FUNCTION_BLOCK FB_2001_cocktail
VAR_INPUT
	execute: BOOL;
END_VAR
VAR
	TIMERDONE: BOOL;
END_VAR

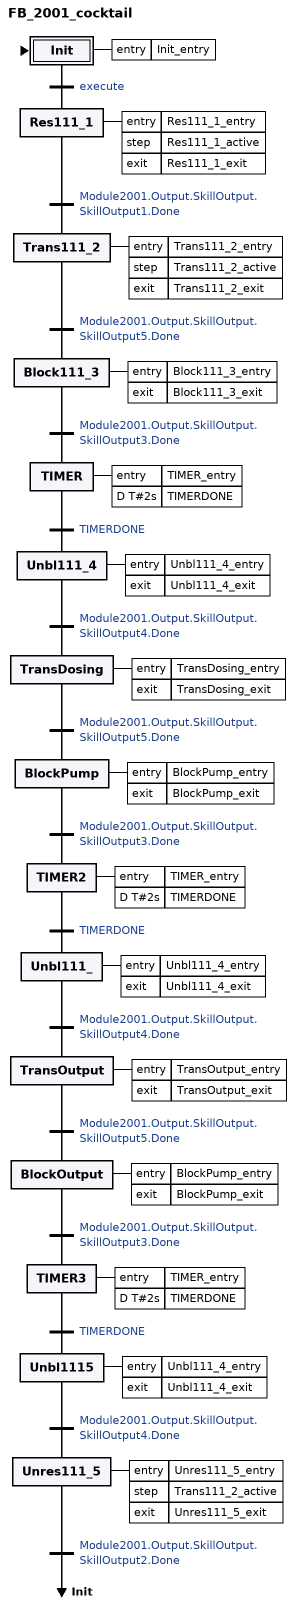
INITIAL_STEP Init:
    Init_entry(P1);  // entry action
END_STEP
TRANSITION FROM Init TO Res111_1
    := execute;
END_TRANSITION
STEP Res111_1:
    Res111_1_entry(P1);  // entry action
    Res111_1_active(N);  // step action
    Res111_1_exit(P0);  // exit action
END_STEP
TRANSITION FROM Res111_1 TO Trans111_2
    := Module2001.Output.SkillOutput.SkillOutput1.Done;
END_TRANSITION
STEP Trans111_2:
    Trans111_2_entry(P1);  // entry action
    Trans111_2_active(N);  // step action
    Trans111_2_exit(P0);  // exit action
END_STEP
TRANSITION FROM Trans111_2 TO Block111_3
    := Module2001.Output.SkillOutput.SkillOutput5.Done;
END_TRANSITION
STEP Block111_3:
    Block111_3_entry(P1);  // entry action
    Block111_3_exit(P0);  // exit action
END_STEP
TRANSITION FROM Block111_3 TO TIMER
    := Module2001.Output.SkillOutput.SkillOutput3.Done;
END_TRANSITION
STEP TIMER:
    TIMER_entry(P1);  // entry action
    TIMERDONE(D, T#2s);
END_STEP
TRANSITION FROM TIMER TO Unbl111_4
    := TIMERDONE;
END_TRANSITION
STEP Unbl111_4:
    Unbl111_4_entry(P1);  // entry action
    Unbl111_4_exit(P0);  // exit action
END_STEP
TRANSITION FROM Unbl111_4 TO TransDosing
    := Module2001.Output.SkillOutput.SkillOutput4.Done;
END_TRANSITION
STEP TransDosing:
    TransDosing_entry(P1);  // entry action
    TransDosing_exit(P0);  // exit action
END_STEP
TRANSITION FROM TransDosing TO BlockPump
    := Module2001.Output.SkillOutput.SkillOutput5.Done;
END_TRANSITION
STEP BlockPump:
    BlockPump_entry(P1);  // entry action
    BlockPump_exit(P0);  // exit action
END_STEP
TRANSITION FROM BlockPump TO TIMER2
    := Module2001.Output.SkillOutput.SkillOutput3.Done;
END_TRANSITION
STEP TIMER2:
    TIMER_entry(P1);  // entry action
    TIMERDONE(D, T#2s);
END_STEP
TRANSITION FROM TIMER2 TO Unbl111_
    := TIMERDONE;
END_TRANSITION
STEP Unbl111_:
    Unbl111_4_entry(P1);  // entry action
    Unbl111_4_exit(P0);  // exit action
END_STEP
TRANSITION FROM Unbl111_ TO TransOutput
    := Module2001.Output.SkillOutput.SkillOutput4.Done;
END_TRANSITION
STEP TransOutput:
    TransOutput_entry(P1);  // entry action
    TransOutput_exit(P0);  // exit action
END_STEP
TRANSITION FROM TransOutput TO BlockOutput
    := Module2001.Output.SkillOutput.SkillOutput5.Done;
END_TRANSITION
STEP BlockOutput:
    BlockPump_entry(P1);  // entry action
    BlockPump_exit(P0);  // exit action
END_STEP
TRANSITION FROM BlockOutput TO TIMER3
    := Module2001.Output.SkillOutput.SkillOutput3.Done;
END_TRANSITION
STEP TIMER3:
    TIMER_entry(P1);  // entry action
    TIMERDONE(D, T#2s);
END_STEP
TRANSITION FROM TIMER3 TO Unbl1115
    := TIMERDONE;
END_TRANSITION
STEP Unbl1115:
    Unbl111_4_entry(P1);  // entry action
    Unbl111_4_exit(P0);  // exit action
END_STEP
TRANSITION FROM Unbl1115 TO Unres111_5
    := Module2001.Output.SkillOutput.SkillOutput4.Done;
END_TRANSITION
STEP Unres111_5:
    Unres111_5_entry(P1);  // entry action
    Trans111_2_active(N);  // step action
    Unres111_5_exit(P0);  // exit action
END_STEP
TRANSITION FROM Unres111_5 TO Init
    := Module2001.Output.SkillOutput.SkillOutput2.Done;
END_TRANSITION

ACTION Unbl111_4_exit:
//unBLOCKIEREN

Module2001.Input.SkillInput.SkillInput4.Execute := FALSE; 
Module2001.Input.SkillInput.SkillInput4.ParameterInput.Parameterinput1.Value := 000; //TaskID
END_ACTION

ACTION Init_entry:
execute := FALSE;
END_ACTION

ACTION Trans111_2_exit:
//TRANSPORTIEREN

Module2001.Input.SkillInput.SkillInput5.Execute := FALSE;
Module2001.Input.SkillInput.SkillInput5.ParameterInput.Parameterinput1.Value := 0; //X-Position
Module2001.Input.SkillInput.SkillInput5.ParameterInput.Parameterinput2.Value := 0; //Z-Position
Module2001.Input.SkillInput.SkillInput5.ParameterInput.Parameterinput3.Value := 0; //Velocity
Module2001.Input.SkillInput.SkillInput5.ParameterInput.Parameterinput4.Value := 0; //Acceleration
END_ACTION

ACTION Unbl111_4_entry:
//unBLOCKIEREN

Module2001.Input.SkillInput.SkillInput4.Execute := TRUE; //FALSE weil timer
Module2001.Input.SkillInput.SkillInput4.ParameterInput.Parameterinput1.Value := 111; //TaskID
END_ACTION

ACTION TIMER_entry:
TIMERDONE := FALSE;
END_ACTION

ACTION TransOutput_exit:

Module2001.Input.SkillInput.SkillInput5.Execute := FALSE;
Module2001.Input.SkillInput.SkillInput5.ParameterInput.Parameterinput1.Value := 0; //X-Position
Module2001.Input.SkillInput.SkillInput5.ParameterInput.Parameterinput2.Value := 0; //Z-Position
Module2001.Input.SkillInput.SkillInput5.ParameterInput.Parameterinput3.Value := 0; //Velocity
Module2001.Input.SkillInput.SkillInput5.ParameterInput.Parameterinput4.Value := 0; //Acceleration
END_ACTION

ACTION TransOutput_entry:
//TRANSPORTIEREN

Module2001.Input.SkillInput.SkillInput5.Execute := TRUE;
Module2001.Input.SkillInput.SkillInput5.ParameterInput.Parameterinput1.Value := 200; //X-Position
Module2001.Input.SkillInput.SkillInput5.ParameterInput.Parameterinput2.Value := 110;//90; //Z-Position
Module2001.Input.SkillInput.SkillInput5.ParameterInput.Parameterinput3.Value := 300; //Velocity
Module2001.Input.SkillInput.SkillInput5.ParameterInput.Parameterinput4.Value := 0; //Acceleration
END_ACTION

ACTION Block111_3_entry:
//BLOCKIEREN

Module2001.Input.SkillInput.SkillInput3.Execute := TRUE;
Module2001.Input.SkillInput.SkillInput3.ParameterInput.Parameterinput1.Value := 111; //TaskID
END_ACTION

ACTION BlockPump_exit:
//BLOCKIEREN

Module2001.Input.SkillInput.SkillInput3.Execute := FALSE;
Module2001.Input.SkillInput.SkillInput3.ParameterInput.Parameterinput1.Value := 0; //TaskID
END_ACTION

ACTION Res111_1_entry:
// Reservieren entry
Module2001.Input.SkillInput.SkillInput1.Execute := TRUE;
Module2001.Input.SkillInput.SkillInput1.ParameterInput.Parameterinput1.Value := 111; //TASKID
END_ACTION

ACTION Res111_1_exit:
// Reservieren entry
Module2001.Input.SkillInput.SkillInput1.Execute := FALSE;
Module2001.Input.SkillInput.SkillInput1.ParameterInput.Parameterinput1.Value := 0; //TASKID
END_ACTION

ACTION Unres111_5_exit:
//unreserve
Module2001.Input.SkillInput.SkillInput2.Execute := FALSE;
Module2001.Input.SkillInput.SkillInput2.ParameterInput.Parameterinput1.Value := 0; //TaskID
END_ACTION

ACTION Res111_1_active:

END_ACTION

ACTION TransDosing_entry:
//TRANSPORTIEREN

Module2001.Input.SkillInput.SkillInput5.Execute := TRUE;
Module2001.Input.SkillInput.SkillInput5.ParameterInput.Parameterinput1.Value := 2200; //X-Position
Module2001.Input.SkillInput.SkillInput5.ParameterInput.Parameterinput2.Value := 20;//90; //Z-Position
Module2001.Input.SkillInput.SkillInput5.ParameterInput.Parameterinput3.Value := 300; //Velocity
Module2001.Input.SkillInput.SkillInput5.ParameterInput.Parameterinput4.Value := 0; //Acceleration
END_ACTION

ACTION Unres111_5_entry:
//unreserve
Module2001.Input.SkillInput.SkillInput2.Execute := TRUE;
Module2001.Input.SkillInput.SkillInput2.ParameterInput.Parameterinput1.Value := 111; //TaskID
END_ACTION

ACTION Block111_3_exit:
//BLOCKIEREN

Module2001.Input.SkillInput.SkillInput3.Execute := FALSE;
Module2001.Input.SkillInput.SkillInput3.ParameterInput.Parameterinput1.Value := 0; //TaskID
END_ACTION

ACTION TransDosing_exit:
//TRANSPORTIEREN

Module2001.Input.SkillInput.SkillInput5.Execute := FALSE;
Module2001.Input.SkillInput.SkillInput5.ParameterInput.Parameterinput1.Value := 0; //X-Position
Module2001.Input.SkillInput.SkillInput5.ParameterInput.Parameterinput2.Value := 0; //Z-Position
Module2001.Input.SkillInput.SkillInput5.ParameterInput.Parameterinput3.Value := 0; //Velocity
Module2001.Input.SkillInput.SkillInput5.ParameterInput.Parameterinput4.Value := 0; //Acceleration
END_ACTION

ACTION BlockPump_entry:
//BLOCKIEREN

Module2001.Input.SkillInput.SkillInput3.Execute := TRUE;
Module2001.Input.SkillInput.SkillInput3.ParameterInput.Parameterinput1.Value := 111; //TaskID
END_ACTION

ACTION Trans111_2_active:

END_ACTION

ACTION Trans111_2_entry:
//TRANSPORTIEREN

Module2001.Input.SkillInput.SkillInput5.Execute := TRUE;
Module2001.Input.SkillInput.SkillInput5.ParameterInput.Parameterinput1.Value := 1300; //X-Position
Module2001.Input.SkillInput.SkillInput5.ParameterInput.Parameterinput2.Value := 0;//90; //Z-Position
Module2001.Input.SkillInput.SkillInput5.ParameterInput.Parameterinput3.Value := 300; //Velocity
Module2001.Input.SkillInput.SkillInput5.ParameterInput.Parameterinput4.Value := 0; //Acceleration
END_ACTION

END_FUNCTION_BLOCK

(* stored: Version 1.1.0.1, ProductVersion 3.1.0.25
   POU FB_2001_cocktail: Id {fb12d113-301a-4245-aa38-124894c67225}
   Action Unbl111_4_exit: Id {045c779b-74c6-429d-8ac6-2006a4087f9e}
   Action Init_entry: Id {16b20ac2-74c8-40a0-866e-d08c2d8e46fb}
   Action Trans111_2_exit: Id {259970b8-6e66-4180-bb57-d26299c5fc3a}
   Action Unbl111_4_entry: Id {3ae651cc-f179-4249-9068-7194905a2fc9}
   Action TIMER_entry: Id {4dfcaa4d-3379-4fdc-8d6a-fade1ffe234a}
   Action TransOutput_exit: Id {5ac9300e-46ee-442c-a788-8e261110346f}
   Action TransOutput_entry: Id {5eb9c766-e66e-4896-87ef-f64a3ff219c0}
   Action Block111_3_entry: Id {6d8d0eec-57e2-4d76-9635-a901ff743fc0}
   Action BlockPump_exit: Id {718a2894-c701-4bba-b7f8-e6bd8b4dcf2f}
   Action Res111_1_entry: Id {82a353d6-c115-46d7-81c2-3b6f92b6c447}
   Action Res111_1_exit: Id {82f2228f-a9f1-43ae-8c81-2093c6b8458f}
   Action Unres111_5_exit: Id {9b5fd2f5-8773-4ede-90f7-bdc4b9c33a12}
   Action Res111_1_active: Id {9c08f0e1-382b-4482-b884-5d6eb34d66e5}
   Action TransDosing_entry: Id {a79ea0cc-4598-4e85-a6ba-ea936f79b119}
   Action Unres111_5_entry: Id {b0a253f1-9981-47de-aa9d-335c5746d1c7}
   Action Block111_3_exit: Id {d2731eb4-a6f4-43a3-a469-64f73ba12412}
   Action TransDosing_exit: Id {d899005f-e4ec-44d4-a806-fdf431382bfc}
   Action BlockPump_entry: Id {db425794-4a2f-4277-8a68-89d52510e50d}
   Action Trans111_2_active: Id {e04fe5bc-972a-4ec9-a131-d8f012ab1859}
   Action Trans111_2_entry: Id {e26d2c96-321d-4ecd-9c72-7de870cb3267} *)
